// TIA Portal V19 export
FUNCTION "PRODUCTION" : Void   // FC41, STL
TITLE = FLOWCOUNTING
{ S7_Optimized_Access := 'TRUE' }
NAME : PRODTANK
VERSION : 0.0
// Programmer Init: 8953-FLA
// 
// Change Log:
// 
// Date        Change                          Updated by
// ------------------------------------------------------
// 19.04.99    1. Edition                      FLA
// 01.06.99    1.1 Counter for mix plant       JOM 8173
// stored: AutoNumber false
BEGIN

NETWORK
TITLE = Move actuel purge setpoint's
      AN    "S0 PRODUCTION TANK";
      R     "DUMMY 1 FILLING";
      R     "DUMMY 2 FILLING";
      R     "T60 OPEN Y0101";
      R     "T61 CLOSE Y0101";
      BEC;
      AN    "T60 OPEN Y0101";
      A     "DUMMY 1 FILLING";
      JC    M003;
      AN    "START FILLING TANK";
      JC    M001;
      R     "START FILLING TANK";
      R     "STOP FILLING TANK";
      AN    "TANK STERILE";
      BEC;
      A     "B01.65";
      O     "HSL0165_Proxy";
      BEC;
      S     "MY0124";
      S     "TIM60";
      S     "DUMMY 1 FILLING";
      BEU;
M003: S     "MY0101";
      R     "TANK CLEAN";
      R     "DUMMY 1 FILLING";
M001: NOP   0;

NETWORK
TITLE = 
      AN    "T61 CLOSE Y0101";
      A     "DUMMY 2 FILLING";
      JC    M004;
      AN    "STOP FILLING TANK";
      JC    M002;
      R     "START FILLING TANK";
      R     "STOP FILLING TANK";
      R     "MY0101";
      S     "TIM61";
      S     "DUMMY 2 FILLING";
      BEU;
M004: R     "MY0124";
      R     "DUMMY 2 FILLING";
M002: NOP   0;
END_FUNCTION
